TYPE Motor :
STRUCT
	Motor_Rated_RPM : REAL;
	Motor_Rated_Hz : REAL;
	Motor_Rated_Power : REAL;
	Motor_Rated_Voltage : REAL;
	Motor_Rated_Current : REAL;
	Motor_CosinePhi : REAL;
END_STRUCT
END_TYPE

(* stored: Version 1.1.0.1, ProductVersion 3.1.4024.12
   DUT Motor: Id {ad7bff48-e75a-4e30-afea-f6d2225a9688} *)
